VAR_GLOBAL
	sRFIDInfo											:	STRING;	// Opis sumy błędów RFID
	bRFIDCheckReset										:	BOOL;	// Reset liczników
	
	iRFIDCheckNumberOfFormsAfterWeighting				:	INT; //Liczba formatek po przeważaniu
	iRFIDCheckNumberOfFormsExecute						:	INT; //Liczba formatek na lini w czasie cyklu
	
	AStRFIDCheck										:	ARRAY [1..100] OF S_RFIDCheck;		
															(*	iNumber				: INT;		//Numer RFID	
																iReaded1			: INT;		//Odczytano z czytnika nr 1 (przed dozownikami) 
																iReaded2			: INT;		//Odczytano z czytnika nr 2	(przed wagami)
																iReaded3			: INT;		//Odczytano z czytnika nr 3	(przed zakrecarka)
																iReaded4			: INT;		//Odczytano z czytnika nr 4 (za zakrecarka)
																iReaded5			: INT;		//Odczytano z czytnika nr 5	(robot)*)
																
	iRFIDCheckDispencerWarning							:	INT;	// Liczba błędnych rejestrów dozowniki
	iRFIDCheckWeightWarning								:	INT;	// Liczba błędnych rejestrów wagi
	iRFIDCheckBeforeScrewerWarning						:	INT;	// Liczba błędnych rejestrów zakrecarki
	iRFIDCheckAfterScrewerWarning						:	INT;	// Liczba błędnych rejestrów test zakrecania
	iRFIDCheckBottleTransferWarning						:	INT;	// Liczba błędnych rejestrów robot
								
END_VAR

(* stored: Version 1.2.0.0, ProductVersion 3.1.4026.13, FileIdentifier ef60fea19a3775b5e75db6bd5d56a2985265ad4f, FileSignature 5354363fd203916ada5ad726ae69a8731c3cfb8d72520a21e449c1664277de6c9563c1470c543e8cf4e7b0cda2966690c6a9fd0ac9367e75f71e34159121d4a9b5eaa3f4f5832486959a31e17fdabdf0c045d6d8c00dba2cb41d3843044004538205daf4e693487e2f8c3b8d7c205c67cac7e06bc6532892a69a1adb69a0b6859007e335161c047d9c65e8857c68553543e7d59642bf4096b73325014b78e8173416a7a2ed31c5bcdbd806f104b076a8e25453d35104a6620297ebde38ce9de9781d454097a9563db0eef9e55620b0f0cfb9f548b800de2d7ff9134b5103c131ee8a7a556fc7ad710069265ba4798cc93f46a9565ae482fe158ff7f5fe508b69
   GVL VIS_RFID: Id {860022f7-34bc-4b41-a0c0-708a6233dafa} *)
